// TIA Portal V20 export
TYPE "typeCmControlNodeCommand"
// stored: Namespace Unit1.Em13
   STRUCT
      jrUnIoadingPnPAxisX : "LER_typeAxisCommand";
      jrUnIoadingPnPAxisZ { S7_SetPoint := 'True'} : "LER_typeAxisCommand";
      jrUnIoadingPnPAxisC { S7_SetPoint := 'True'} : "LER_typeAxisCommand";
      jrUnIoadingPnPClamp { S7_SetPoint := 'True'} : "LER_typeTwoWayActCommand";
   END_STRUCT;
END_TYPE
